// Interface for logging methods which can be called in user code.
INTERFACE I_Logger

METHOD LogCritical
VAR_INPUT
  message : T_MessageString; 
END_VAR
END_METHOD

METHOD LogError
VAR_INPUT
  message : T_MessageString; 
END_VAR
END_METHOD

METHOD LogInfo
VAR_INPUT
  message : T_MessageString; 
END_VAR
END_METHOD

METHOD LogVerbose
VAR_INPUT
  message : T_MessageString; 
END_VAR
END_METHOD

METHOD LogWarning
VAR_INPUT
  message : T_MessageString; 
END_VAR
END_METHOD

END_INTERFACE

(* stored: Version 1.1.0.1, ProductVersion 3.1.4024.12
   Itf I_Logger: Id {cc905d47-10eb-0e51-37da-280142df90f2}
   Method LogCritical: Id {c1e8cb14-7a09-0680-2f7e-0bbd0d102f2f}
   Method LogError: Id {1c0fd136-d0b9-02ed-3f94-f5133f04c6e3}
   Method LogInfo: Id {87c86887-5e85-0549-2419-4a17a416df33}
   Method LogVerbose: Id {e7847836-d92c-064f-0687-2c232ac0e658}
   Method LogWarning: Id {f4efeaae-1adc-0e37-22b6-ca2ee4018346} *)
